// TIA Portal V21 export
// export: Created 2026-09-06T16:13:42.819562Z, ExportSetting WithDefaults, DisplayName Totally Integrated Automation Portal, DisplayVersion V21 Hotfix 1, DisplayName STEP 7 Professional, DisplayVersion V21, DisplayName STEP 7 CFC, DisplayVersion V21, DisplayName STEP 7 Safety, DisplayVersion V21, DisplayName Tech WebApplication, DisplayVersion V21, DisplayName WinCC Basic/Comfort/Advanced, DisplayVersion V21, DisplayName SIMATIC Visualization Architect, DisplayVersion V21, DisplayName WinCC Unified, DisplayVersion V21, DisplayName SIMATIC Visualization Architect, DisplayVersion V21
VAR_GLOBAL   // PLC tag table "Saidas_CPU_Local"
   KM1 AT %Q0.0 : Bool;   // Contactor de Processo do Motor M1 (Tapete 1)
   KM2 AT %Q0.1 : Bool;   // Contactor de Processo do Motor M2 (Tapete 2)
   KM3 AT %Q0.2 : Bool;   // Contactor de Processo do Motor M3 (Tapete 3)
   KM4 AT %Q0.3 : Bool;   // Contactor de Processo do Motor M4 (Tapete 4)
   KM5 AT %Q0.4 : Bool;   // Contactor de Processo do Motor M5 (Tapete 5)
   START_SS_M6 AT %Q0.5 : Bool;   // Sinal de Habilitacao / Start da Soft Starter (Bomba M6)
   Y1_AVANCA AT %Q0.6 : Bool;   // Eletrovalvula de Avanco do Cilindro Hidraulico
   Y2_RECUA AT %Q0.7 : Bool;   // Eletrovalvula de Recuo do Cilindro Hidraulico
   H1_VERDE AT %Q1.0 : Bool;   // Sinalizador Luminoso Verde: Linha em Funcionamento / Automatico
   H2_AMARELO AT %Q1.1 : Bool;   // Sinalizador Luminoso Amarelo: Estado de Prontidao / Standby
END_VAR
